TYPE T_PCM_Filename : T_MaxString;
END_TYPE

(* stored: Version 1.1.0.1
   DUT T_PCM_Filename: Id {cf1008ad-6240-4701-b38c-edaa930ced58} *)
